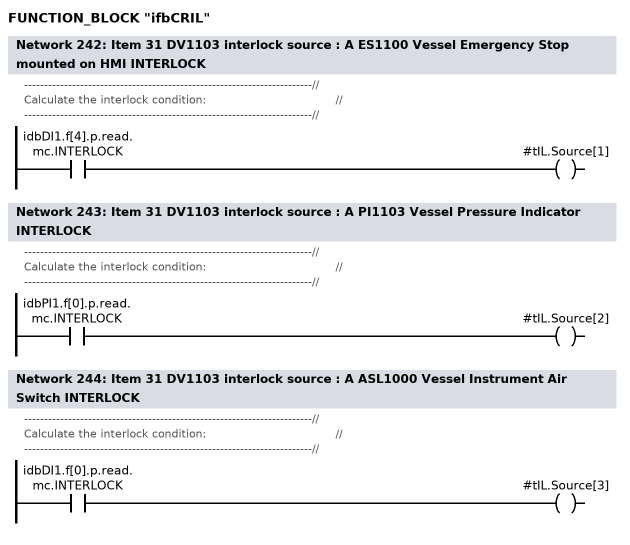
    A idbDI1.f[4].p.read.mc.INTERLOCK;
    = #tIL.Source[1];

NETWORK
TITLE = Item 31 DV1103 interlock source : A PI1103 Vessel Pressure Indicator INTERLOCK
    //------------------------------------------------------------------------//
    // Calculate the interlock condition:                                     //
    //------------------------------------------------------------------------//
    A idbPI1.f[0].p.read.mc.INTERLOCK;
    = #tIL.Source[2];

NETWORK
TITLE = Item 31 DV1103 interlock source : A ASL1000 Vessel Instrument Air Switch INTERLOCK
    //------------------------------------------------------------------------//
    // Calculate the interlock condition:                                     //
    //------------------------------------------------------------------------//
    A idbDI1.f[0].p.read.mc.INTERLOCK;
    = #tIL.Source[3];

NETWORK
TITLE = Item 31 DV1103 interlock source : AN ZSC1101 Vessel Manway Closed Indicator CLOSED
    //------------------------------------------------------------------------//
    // Calculate the interlock condition:                                     //
    //------------------------------------------------------------------------//
    AN(;
    L "idbZSC1".f[0].p.read.mc.STATE;
    L "dbCONST".BLK.ZSC1.STATE.CLOSED;
    ==I;
    );
    = #tIL.Source[4];

NETWORK
TITLE = Item 31 DV1103 interlock source : A ES1101 Mx Emergency Stop mounted on M1/M2 Shared HMI INTERLOCK
    //------------------------------------------------------------------------//
    // Calculate the interlock condition:                                     //
    //------------------------------------------------------------------------//
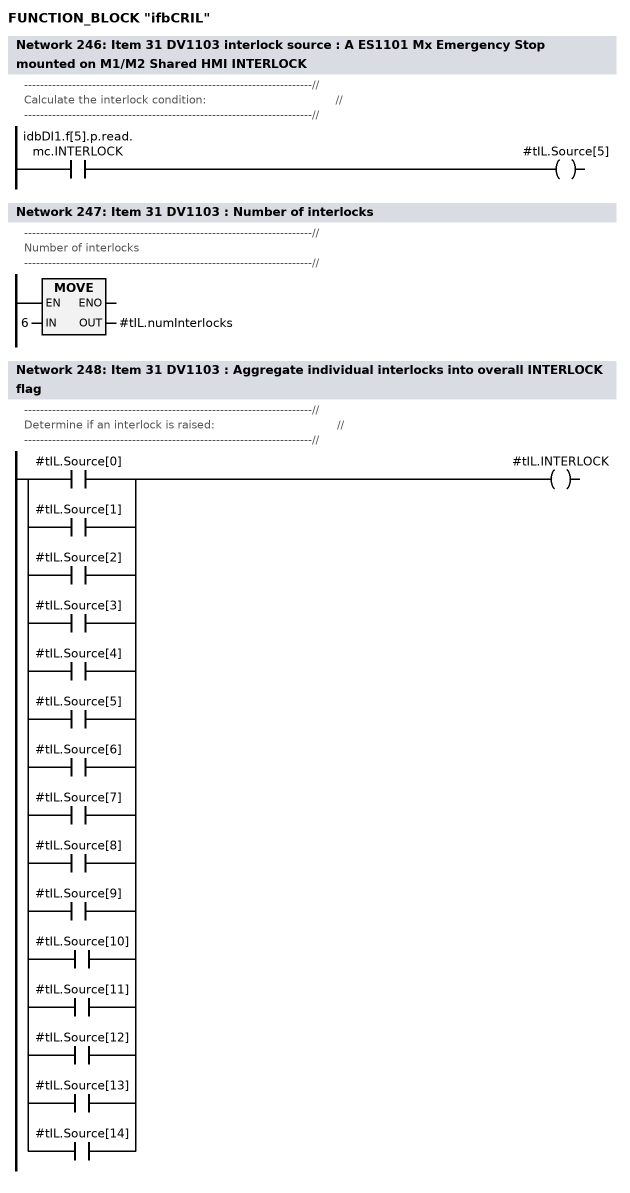
    A idbDI1.f[5].p.read.mc.INTERLOCK;
    = #tIL.Source[5];


NETWORK
TITLE = Item 31 DV1103 : Number of interlocks
    //------------------------------------------------------------------------//
    // Number of interlocks
    //------------------------------------------------------------------------//
    L 6;
    T #tIL.numInterlocks;

NETWORK
TITLE = Item 31 DV1103 : Aggregate individual interlocks into overall INTERLOCK flag
    //------------------------------------------------------------------------//
    // Determine if an interlock is raised:                                   //
    //------------------------------------------------------------------------//
    O #tIL.Source[0];
    O #tIL.Source[1];
    O #tIL.Source[2];
    O #tIL.Source[3];
    O #tIL.Source[4];
    O #tIL.Source[5];
    O #tIL.Source[6];
    O #tIL.Source[7];
    O #tIL.Source[8];
    O #tIL.Source[9];
    O #tIL.Source[10];
    O #tIL.Source[11];
    O #tIL.Source[12];
    O #tIL.Source[13];
    O #tIL.Source[14];
    = #tIL.INTERLOCK;

NETWORK
TITLE = Item 31 DV1103 : Update the instance data
    //------------------------------------------------------------------------//
    // Update the instance DB with the calculated interlock flags:            //
    //------------------------------------------------------------------------//
    CALL MOVE
    {value_type := 'Variant'}
    (   IN                   := #tIL ,
        OUT                  := #p[31]
    );

NETWORK
TITLE = Item 32 DV1105 : LP CA Supply Valve initialise variables
    //------------------------------------------------------------------------//
    // CRITICAL INTERLOCK   CRITICAL INTERLOCK   CRITICAL INTERLOCK   CRITICA //
    // CRITICAL INTERLOCK   CRITICAL INTERLOCK   CRITICAL INTERLOCK   CRITICA //
    //                                                                        //
    // Clear the interlock flag:                                              //
    //------------------------------------------------------------------------//
    A "alwaysLow";
    = #tIL.INTERLOCK;

    //------------------------------------------------------------------------//
    // Clear all interlock values to initialise them to off:                  //
    //------------------------------------------------------------------------//
    CALL FILL_BLK
    {value_type := 'Bool', count_type := 'UInt'}
    (   IN                   := 0 ,
        COUNT                := 15 ,
        OUT                  := #tIL.Source[0]
    );


NETWORK
TITLE = Item 32 DV1105 interlock source : A RD1101 Vessel Burst Disc ALARM
    //------------------------------------------------------------------------//
    // Calculate the interlock condition:                                     //
    //------------------------------------------------------------------------//
    A idbDI1.f[13].p.read.mc.INTERLOCK;
    = #tIL.Source[0];

NETWORK
TITLE = Item 32 DV1105 interlock source : A ES1100 Vessel Emergency Stop mounted on HMI INTERLOCK
    //------------------------------------------------------------------------//
    // Calculate the interlock condition:                                     //
    //------------------------------------------------------------------------//
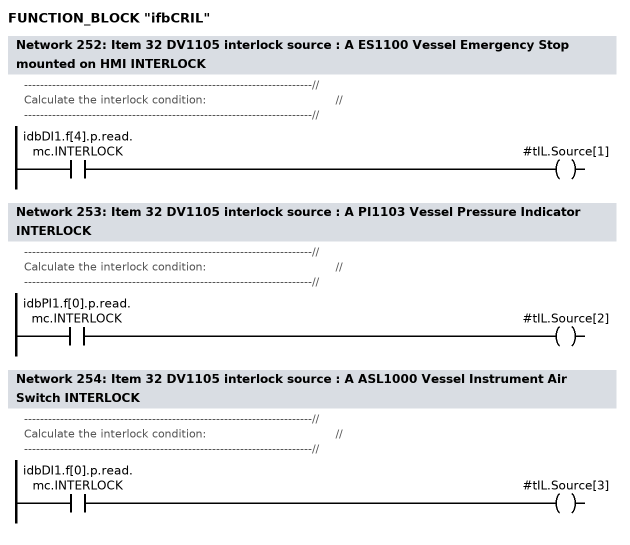
    A idbDI1.f[4].p.read.mc.INTERLOCK;
    = #tIL.Source[1];

NETWORK
TITLE = Item 32 DV1105 interlock source : A PI1103 Vessel Pressure Indicator INTERLOCK
    //------------------------------------------------------------------------//
    // Calculate the interlock condition:                                     //
    //------------------------------------------------------------------------//
    A idbPI1.f[0].p.read.mc.INTERLOCK;
    = #tIL.Source[2];

NETWORK
TITLE = Item 32 DV1105 interlock source : A ASL1000 Vessel Instrument Air Switch INTERLOCK
    //------------------------------------------------------------------------//
    // Calculate the interlock condition:                                     //
    //------------------------------------------------------------------------//
    A idbDI1.f[0].p.read.mc.INTERLOCK;
    = #tIL.Source[3];

NETWORK
TITLE = Item 32 DV1105 interlock source : AN ZSC1101 Vessel Manway Closed Indicator CLOSED
    //------------------------------------------------------------------------//
    // Calculate the interlock condition:                                     //
    //------------------------------------------------------------------------//
    AN(;
    L "idbZSC1".f[0].p.read.mc.STATE;
    L "dbCONST".BLK.ZSC1.STATE.CLOSED;
    ==I;
    );
    = #tIL.Source[4];

NETWORK
TITLE = Item 32 DV1105 interlock source : A ES1101 Mx Emergency Stop mounted on M1/M2 Shared HMI INTERLOCK
    //------------------------------------------------------------------------//
    // Calculate the interlock condition:                                     //
    //------------------------------------------------------------------------//
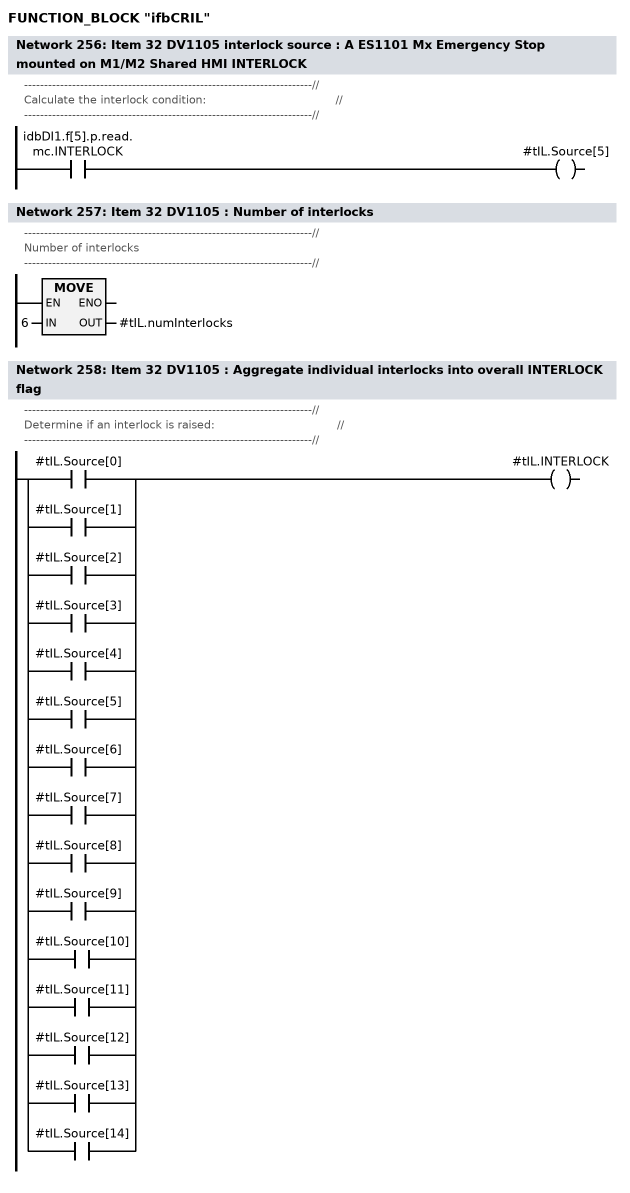
    A idbDI1.f[5].p.read.mc.INTERLOCK;
    = #tIL.Source[5];


NETWORK
TITLE = Item 32 DV1105 : Number of interlocks
    //------------------------------------------------------------------------//
    // Number of interlocks
    //------------------------------------------------------------------------//
    L 6;
    T #tIL.numInterlocks;

NETWORK
TITLE = Item 32 DV1105 : Aggregate individual interlocks into overall INTERLOCK flag
    //------------------------------------------------------------------------//
    // Determine if an interlock is raised:                                   //
    //------------------------------------------------------------------------//
    O #tIL.Source[0];
    O #tIL.Source[1];
    O #tIL.Source[2];
    O #tIL.Source[3];
    O #tIL.Source[4];
    O #tIL.Source[5];
    O #tIL.Source[6];
    O #tIL.Source[7];
    O #tIL.Source[8];
    O #tIL.Source[9];
    O #tIL.Source[10];
    O #tIL.Source[11];
    O #tIL.Source[12];
    O #tIL.Source[13];
    O #tIL.Source[14];
    = #tIL.INTERLOCK;

NETWORK
TITLE = Item 32 DV1105 : Update the instance data
    //------------------------------------------------------------------------//
    // Update the instance DB with the calculated interlock flags:            //
    //------------------------------------------------------------------------//
    CALL MOVE
    {value_type := 'Variant'}
    (   IN                   := #tIL ,
        OUT                  := #p[32]
    );

NETWORK
TITLE = Item 33 DV1107 : Vacuum valve initialise variables
    //------------------------------------------------------------------------//
    // CRITICAL INTERLOCK   CRITICAL INTERLOCK   CRITICAL INTERLOCK   CRITICA //
    // CRITICAL INTERLOCK   CRITICAL INTERLOCK   CRITICAL INTERLOCK   CRITICA //
    //                                                                        //
    // Clear the interlock flag:                                              //
    //------------------------------------------------------------------------//
    A "alwaysLow";
    = #tIL.INTERLOCK;

    //------------------------------------------------------------------------//
    // Clear all interlock values to initialise them to off:                  //
    //------------------------------------------------------------------------//
    CALL FILL_BLK
    {value_type := 'Bool', count_type := 'UInt'}
    (   IN                   := 0 ,
        COUNT                := 15 ,
        OUT                  := #tIL.Source[0]
    );


NETWORK
TITLE = Item 33 DV1107 interlock source : A RD1101 Vessel Burst Disc ALARM
    //------------------------------------------------------------------------//
    // Calculate the interlock condition:                                     //
    //------------------------------------------------------------------------//
    A idbDI1.f[13].p.read.mc.INTERLOCK;
    = #tIL.Source[0];

NETWORK
TITLE = Item 33 DV1107 interlock source : A ES1100 Vessel Emergency Stop mounted on HMI INTERLOCK
    //------------------------------------------------------------------------//
    // Calculate the interlock condition:                                     //
    //------------------------------------------------------------------------//
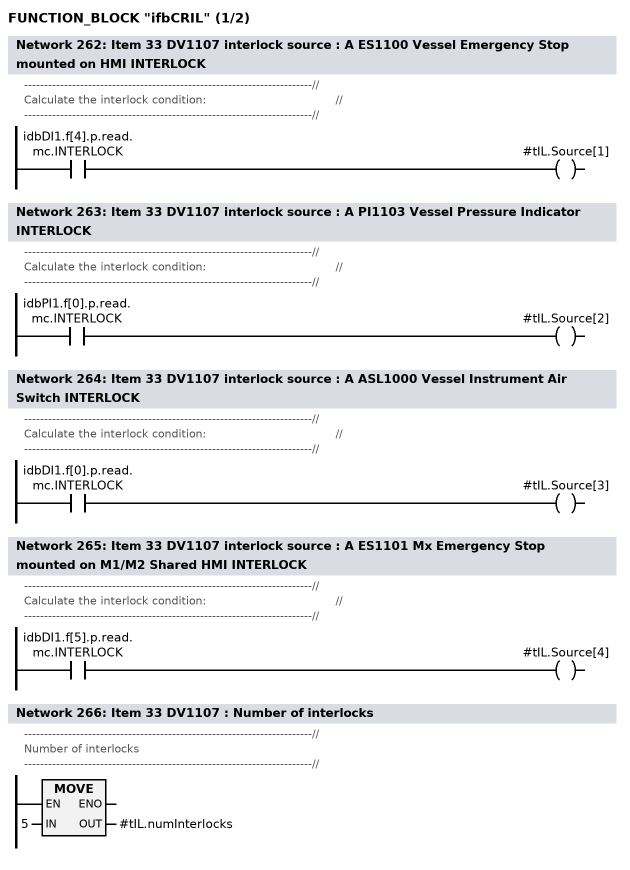
    A idbDI1.f[4].p.read.mc.INTERLOCK;
    = #tIL.Source[1];

NETWORK
TITLE = Item 33 DV1107 interlock source : A PI1103 Vessel Pressure Indicator INTERLOCK
    //------------------------------------------------------------------------//
    // Calculate the interlock condition:                                     //
    //------------------------------------------------------------------------//
    A idbPI1.f[0].p.read.mc.INTERLOCK;
    = #tIL.Source[2];

NETWORK
TITLE = Item 33 DV1107 interlock source : A ASL1000 Vessel Instrument Air Switch INTERLOCK
    //------------------------------------------------------------------------//
    // Calculate the interlock condition:                                     //
    //------------------------------------------------------------------------//
    A idbDI1.f[0].p.read.mc.INTERLOCK;
    = #tIL.Source[3];

NETWORK
TITLE = Item 33 DV1107 interlock source : A ES1101 Mx Emergency Stop mounted on M1/M2 Shared HMI INTERLOCK
    //------------------------------------------------------------------------//
    // Calculate the interlock condition:                                     //
    //------------------------------------------------------------------------//
    A idbDI1.f[5].p.read.mc.INTERLOCK;
    = #tIL.Source[4];


NETWORK
TITLE = Item 33 DV1107 : Number of interlocks
    //------------------------------------------------------------------------//
    // Number of interlocks
    //------------------------------------------------------------------------//
    L 5;
    T #tIL.numInterlocks;

NETWORK
TITLE = Item 33 DV1107 : Aggregate individual interlocks into overall INTERLOCK flag
    //------------------------------------------------------------------------//
    // Determine if an interlock is raised:                                   //
    //------------------------------------------------------------------------//
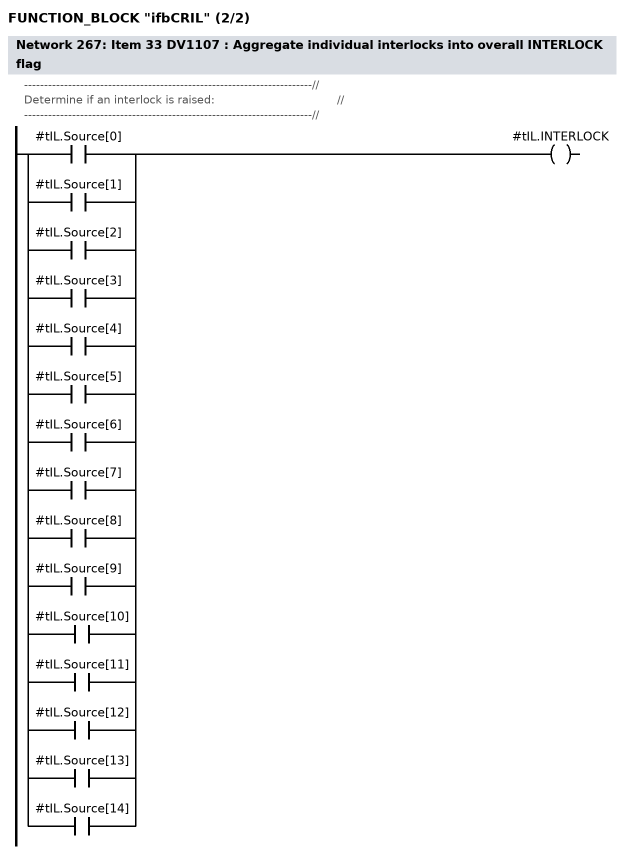
    O #tIL.Source[0];
    O #tIL.Source[1];
    O #tIL.Source[2];
    O #tIL.Source[3];
    O #tIL.Source[4];
    O #tIL.Source[5];
    O #tIL.Source[6];
    O #tIL.Source[7];
    O #tIL.Source[8];
    O #tIL.Source[9];
    O #tIL.Source[10];
    O #tIL.Source[11];
    O #tIL.Source[12];
    O #tIL.Source[13];
    O #tIL.Source[14];
    = #tIL.INTERLOCK;

NETWORK
TITLE = Item 33 DV1107 : Update the instance data
    //------------------------------------------------------------------------//
    // Update the instance DB with the calculated interlock flags:            //
    //------------------------------------------------------------------------//
    CALL MOVE
    {value_type := 'Variant'}
    (   IN                   := #tIL ,
        OUT                  := #p[33]
    );

NETWORK
TITLE = Item 34 DV1109 : PS Supply for WFI Loop initialise variables
    //------------------------------------------------------------------------//
    // CRITICAL INTERLOCK   CRITICAL INTERLOCK   CRITICAL INTERLOCK   CRITICA //
    // CRITICAL INTERLOCK   CRITICAL INTERLOCK   CRITICAL INTERLOCK   CRITICA //
    //                                                                        //
    // Clear the interlock flag:                                              //
    //------------------------------------------------------------------------//
    A "alwaysLow";
    = #tIL.INTERLOCK;

    //------------------------------------------------------------------------//
    // Clear all interlock values to initialise them to off:                  //
    //------------------------------------------------------------------------//
    CALL FILL_BLK
    {value_type := 'Bool', count_type := 'UInt'}
    (   IN                   := 0 ,
        COUNT                := 15 ,
        OUT                  := #tIL.Source[0]
    );


NETWORK
TITLE = Item 34 DV1109 interlock source : ON ZSC1107 Vessel inlet line Flowpath Indicator IN   ON ZSC1103 Vessel WFI Supply Flowpath Indicator IN
    //------------------------------------------------------------------------//
    // Calculate the interlock condition:                                     //
    //------------------------------------------------------------------------//
    ON(;
    L "idbZSC2".f[2].p.read.mc.STATE;
    L "dbCONST".BLK.ZSC2.STATE.IN;
    ==I;
    );
ON(;
    L "idbZSC2".f[0].p.read.mc.STATE;
    L "dbCONST".BLK.ZSC2.STATE.IN;
    ==I;
    );
    = #tIL.Source[0];

NETWORK
TITLE = Item 34 DV1109 interlock source : A DV1111 Vessel WFI Supply Valve OPENED
    //------------------------------------------------------------------------//
    // Calculate the interlock condition:                                     //
    //------------------------------------------------------------------------//
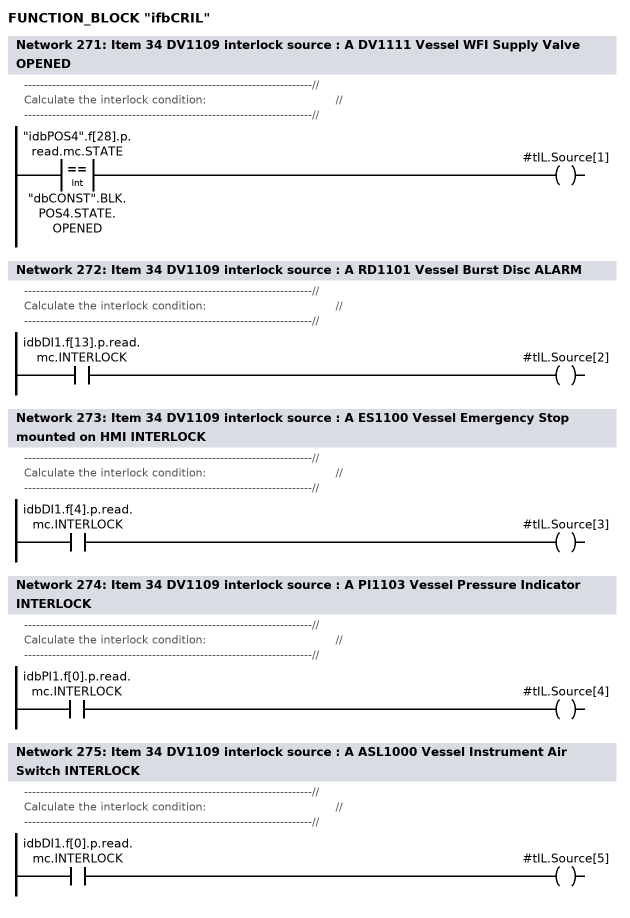
    A(;
    L "idbPOS4".f[28].p.read.mc.STATE;
    L "dbCONST".BLK.POS4.STATE.OPENED;
    ==I;
    );
    = #tIL.Source[1];

NETWORK
TITLE = Item 34 DV1109 interlock source : A RD1101 Vessel Burst Disc ALARM
    //------------------------------------------------------------------------//
    // Calculate the interlock condition:                                     //
    //------------------------------------------------------------------------//
    A idbDI1.f[13].p.read.mc.INTERLOCK;
    = #tIL.Source[2];

NETWORK
TITLE = Item 34 DV1109 interlock source : A ES1100 Vessel Emergency Stop mounted on HMI INTERLOCK
    //------------------------------------------------------------------------//
    // Calculate the interlock condition:                                     //
    //------------------------------------------------------------------------//
    A idbDI1.f[4].p.read.mc.INTERLOCK;
    = #tIL.Source[3];

NETWORK
TITLE = Item 34 DV1109 interlock source : A PI1103 Vessel Pressure Indicator INTERLOCK
    //------------------------------------------------------------------------//
    // Calculate the interlock condition:                                     //
    //------------------------------------------------------------------------//
    A idbPI1.f[0].p.read.mc.INTERLOCK;
    = #tIL.Source[4];

NETWORK
TITLE = Item 34 DV1109 interlock source : A ASL1000 Vessel Instrument Air Switch INTERLOCK
    //------------------------------------------------------------------------//
    // Calculate the interlock condition:                                     //
    //------------------------------------------------------------------------//
    A idbDI1.f[0].p.read.mc.INTERLOCK;
    = #tIL.Source[5];

NETWORK
TITLE = Item 34 DV1109 interlock source : AN ZSC1101 Vessel Manway Closed Indicator CLOSED
    //------------------------------------------------------------------------//
    // Calculate the interlock condition:                                     //
    //------------------------------------------------------------------------//
    AN(;
    L "idbZSC1".f[0].p.read.mc.STATE;
    L "dbCONST".BLK.ZSC1.STATE.CLOSED;
    ==I;
    );
    = #tIL.Source[6];

NETWORK
TITLE = Item 34 DV1109 interlock source : O MI1101 Mx Mass Indicator High High Alarm ALARM_HH   ON MI1101 Mx Mass Indicator Bad DQ DQ
    //------------------------------------------------------------------------//
    // Calculate the interlock condition:                                     //
    //------------------------------------------------------------------------//
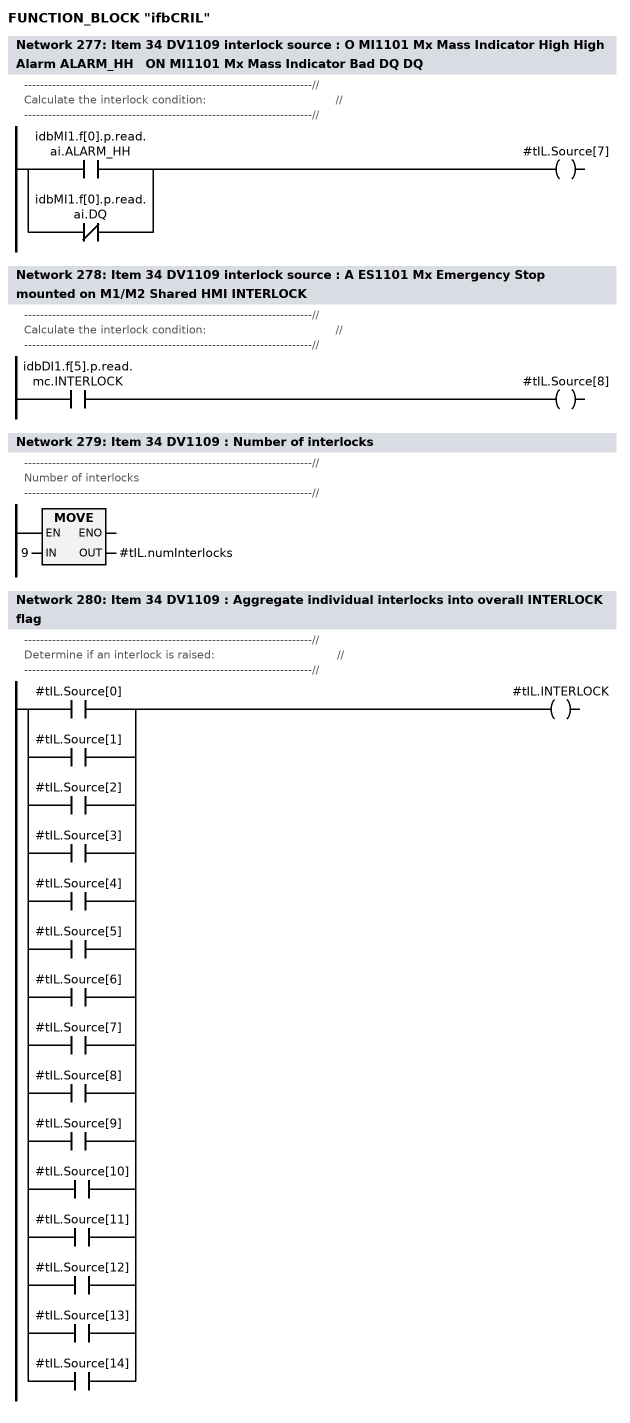
    O idbMI1.f[0].p.read.ai.ALARM_HH;
ON idbMI1.f[0].p.read.ai.DQ;
    = #tIL.Source[7];

NETWORK
TITLE = Item 34 DV1109 interlock source : A ES1101 Mx Emergency Stop mounted on M1/M2 Shared HMI INTERLOCK
    //------------------------------------------------------------------------//
    // Calculate the interlock condition:                                     //
    //------------------------------------------------------------------------//
    A idbDI1.f[5].p.read.mc.INTERLOCK;
    = #tIL.Source[8];


NETWORK
TITLE = Item 34 DV1109 : Number of interlocks
    //------------------------------------------------------------------------//
    // Number of interlocks
    //------------------------------------------------------------------------//
    L 9;
    T #tIL.numInterlocks;

NETWORK
TITLE = Item 34 DV1109 : Aggregate individual interlocks into overall INTERLOCK flag
    //------------------------------------------------------------------------//
    // Determine if an interlock is raised:                                   //
    //------------------------------------------------------------------------//
    O #tIL.Source[0];
    O #tIL.Source[1];
    O #tIL.Source[2];
    O #tIL.Source[3];
    O #tIL.Source[4];
    O #tIL.Source[5];
    O #tIL.Source[6];
    O #tIL.Source[7];
    O #tIL.Source[8];
    O #tIL.Source[9];
    O #tIL.Source[10];
    O #tIL.Source[11];
    O #tIL.Source[12];
    O #tIL.Source[13];
    O #tIL.Source[14];
    = #tIL.INTERLOCK;

NETWORK
TITLE = Item 34 DV1109 : Update the instance data
    //------------------------------------------------------------------------//
    // Update the instance DB with the calculated interlock flags:            //
    //------------------------------------------------------------------------//
    CALL MOVE
    {value_type := 'Variant'}
    (   IN                   := #tIL ,
        OUT                  := #p[34]
    );

NETWORK
TITLE = Item 35 DV1111 : WFI Supply Valve initialise variables
    //------------------------------------------------------------------------//
    // CRITICAL INTERLOCK   CRITICAL INTERLOCK   CRITICAL INTERLOCK   CRITICA //
    // CRITICAL INTERLOCK   CRITICAL INTERLOCK   CRITICAL INTERLOCK   CRITICA //
    //                                                                        //
    // Clear the interlock flag:                                              //
    //------------------------------------------------------------------------//
    A "alwaysLow";
    = #tIL.INTERLOCK;

    //------------------------------------------------------------------------//
    // Clear all interlock values to initialise them to off:                  //
    //------------------------------------------------------------------------//
    CALL FILL_BLK
    {value_type := 'Bool', count_type := 'UInt'}
    (   IN                   := 0 ,
        COUNT                := 15 ,
        OUT                  := #tIL.Source[0]
    );


NETWORK
TITLE = Item 35 DV1111 interlock source : ON ZSC1107 Vessel inlet line Flowpath Indicator IN   ON ZSC1103 Vessel WFI Supply Flowpath Indicator IN
    //------------------------------------------------------------------------//
    // Calculate the interlock condition:                                     //
    //------------------------------------------------------------------------//
    ON(;
    L "idbZSC2".f[2].p.read.mc.STATE;
    L "dbCONST".BLK.ZSC2.STATE.IN;
    ==I;
    );
ON(;
    L "idbZSC2".f[0].p.read.mc.STATE;
    L "dbCONST".BLK.ZSC2.STATE.IN;
    ==I;
    );
    = #tIL.Source[0];

NETWORK
TITLE = Item 35 DV1111 interlock source : A DV1109 Vessel PS Supply for WFI Loop OPENED
    //------------------------------------------------------------------------//
    // Calculate the interlock condition:                                     //
    //------------------------------------------------------------------------//
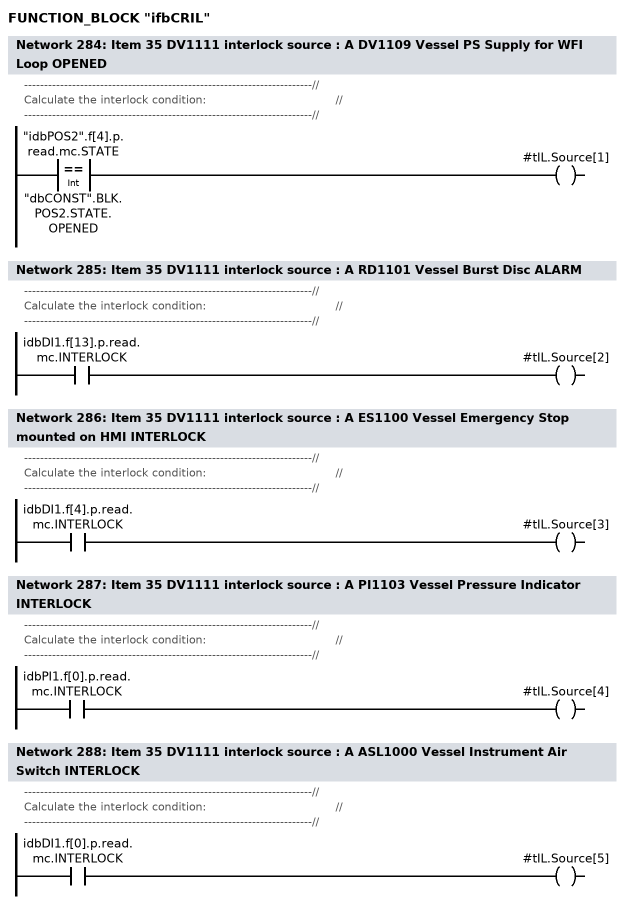
    A(;
    L "idbPOS2".f[4].p.read.mc.STATE;
    L "dbCONST".BLK.POS2.STATE.OPENED;
    ==I;
    );
    = #tIL.Source[1];

NETWORK
TITLE = Item 35 DV1111 interlock source : A RD1101 Vessel Burst Disc ALARM
    //------------------------------------------------------------------------//
    // Calculate the interlock condition:                                     //
    //------------------------------------------------------------------------//
    A idbDI1.f[13].p.read.mc.INTERLOCK;
    = #tIL.Source[2];

NETWORK
TITLE = Item 35 DV1111 interlock source : A ES1100 Vessel Emergency Stop mounted on HMI INTERLOCK
    //------------------------------------------------------------------------//
    // Calculate the interlock condition:                                     //
    //------------------------------------------------------------------------//
    A idbDI1.f[4].p.read.mc.INTERLOCK;
    = #tIL.Source[3];

NETWORK
TITLE = Item 35 DV1111 interlock source : A PI1103 Vessel Pressure Indicator INTERLOCK
    //------------------------------------------------------------------------//
    // Calculate the interlock condition:                                     //
    //------------------------------------------------------------------------//
    A idbPI1.f[0].p.read.mc.INTERLOCK;
    = #tIL.Source[4];

NETWORK
TITLE = Item 35 DV1111 interlock source : A ASL1000 Vessel Instrument Air Switch INTERLOCK
    //------------------------------------------------------------------------//
    // Calculate the interlock condition:                                     //
    //------------------------------------------------------------------------//
    A idbDI1.f[0].p.read.mc.INTERLOCK;
    = #tIL.Source[5];

NETWORK
TITLE = Item 35 DV1111 interlock source : AN ZSC1101 Vessel Manway Closed Indicator CLOSED
    //------------------------------------------------------------------------//
    // Calculate the interlock condition:                                     //
    //------------------------------------------------------------------------//
    AN(;
    L "idbZSC1".f[0].p.read.mc.STATE;
    L "dbCONST".BLK.ZSC1.STATE.CLOSED;
    ==I;
    );
    = #tIL.Source[6];

NETWORK
TITLE = Item 35 DV1111 interlock source : O MI1101 Mx Mass Indicator High High Alarm ALARM_HH   ON MI1101 Mx Mass Indicator Bad DQ DQ
    //------------------------------------------------------------------------//
    // Calculate the interlock condition:                                     //
    //------------------------------------------------------------------------//
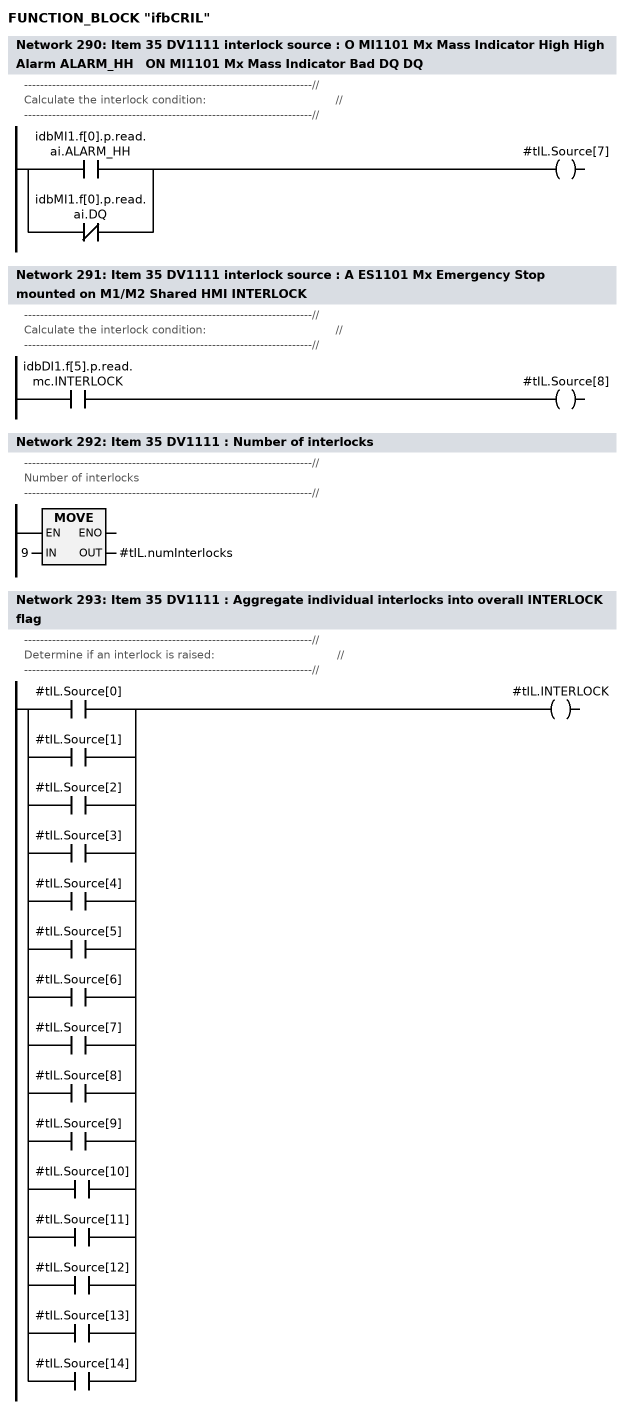
    O idbMI1.f[0].p.read.ai.ALARM_HH;
ON idbMI1.f[0].p.read.ai.DQ;
    = #tIL.Source[7];

NETWORK
TITLE = Item 35 DV1111 interlock source : A ES1101 Mx Emergency Stop mounted on M1/M2 Shared HMI INTERLOCK
    //------------------------------------------------------------------------//
    // Calculate the interlock condition:                                     //
    //------------------------------------------------------------------------//
    A idbDI1.f[5].p.read.mc.INTERLOCK;
    = #tIL.Source[8];


NETWORK
TITLE = Item 35 DV1111 : Number of interlocks
    //------------------------------------------------------------------------//
    // Number of interlocks
    //------------------------------------------------------------------------//
    L 9;
    T #tIL.numInterlocks;

NETWORK
TITLE = Item 35 DV1111 : Aggregate individual interlocks into overall INTERLOCK flag
    //------------------------------------------------------------------------//
    // Determine if an interlock is raised:                                   //
    //------------------------------------------------------------------------//
    O #tIL.Source[0];
    O #tIL.Source[1];
    O #tIL.Source[2];
    O #tIL.Source[3];
    O #tIL.Source[4];
    O #tIL.Source[5];
    O #tIL.Source[6];
    O #tIL.Source[7];
    O #tIL.Source[8];
    O #tIL.Source[9];
    O #tIL.Source[10];
    O #tIL.Source[11];
    O #tIL.Source[12];
    O #tIL.Source[13];
    O #tIL.Source[14];
    = #tIL.INTERLOCK;

NETWORK
TITLE = Item 35 DV1111 : Update the instance data
    //------------------------------------------------------------------------//
    // Update the instance DB with the calculated interlock flags:            //
    //------------------------------------------------------------------------//
    CALL MOVE
    {value_type := 'Variant'}
    (   IN                   := #tIL ,
        OUT                  := #p[35]
    );

NETWORK
TITLE = Item 36 DV1113 : PW Supply Valve initialise variables
    //------------------------------------------------------------------------//
    // CRITICAL INTERLOCK   CRITICAL INTERLOCK   CRITICAL INTERLOCK   CRITICA //
    // CRITICAL INTERLOCK   CRITICAL INTERLOCK   CRITICAL INTERLOCK   CRITICA //
    //                                                                        //
    // Clear the interlock flag:                                              //
    //------------------------------------------------------------------------//
    A "alwaysLow";
    = #tIL.INTERLOCK;

    //------------------------------------------------------------------------//
    // Clear all interlock values to initialise them to off:                  //
    //------------------------------------------------------------------------//
    CALL FILL_BLK
    {value_type := 'Bool', count_type := 'UInt'}
    (   IN                   := 0 ,
        COUNT                := 15 ,
        OUT                  := #tIL.Source[0]
    );


NETWORK
TITLE = Item 36 DV1113 interlock source : ON ZSC1107 Vessel inlet line Flowpath Indicator IN   ON ZSC1105 Vessel PW Supply Flowpath Indicator IN
    //------------------------------------------------------------------------//
    // Calculate the interlock condition:                                     //
    //------------------------------------------------------------------------//
    ON(;
    L "idbZSC2".f[2].p.read.mc.STATE;
    L "dbCONST".BLK.ZSC2.STATE.IN;
    ==I;
    );
ON(;
    L "idbZSC2".f[1].p.read.mc.STATE;
    L "dbCONST".BLK.ZSC2.STATE.IN;
    ==I;
    );
    = #tIL.Source[0];

NETWORK
TITLE = Item 36 DV1113 interlock source : A DV1115 Vessel PS Supply for PW Loop OPENED
    //------------------------------------------------------------------------//
    // Calculate the interlock condition:                                     //
    //------------------------------------------------------------------------//
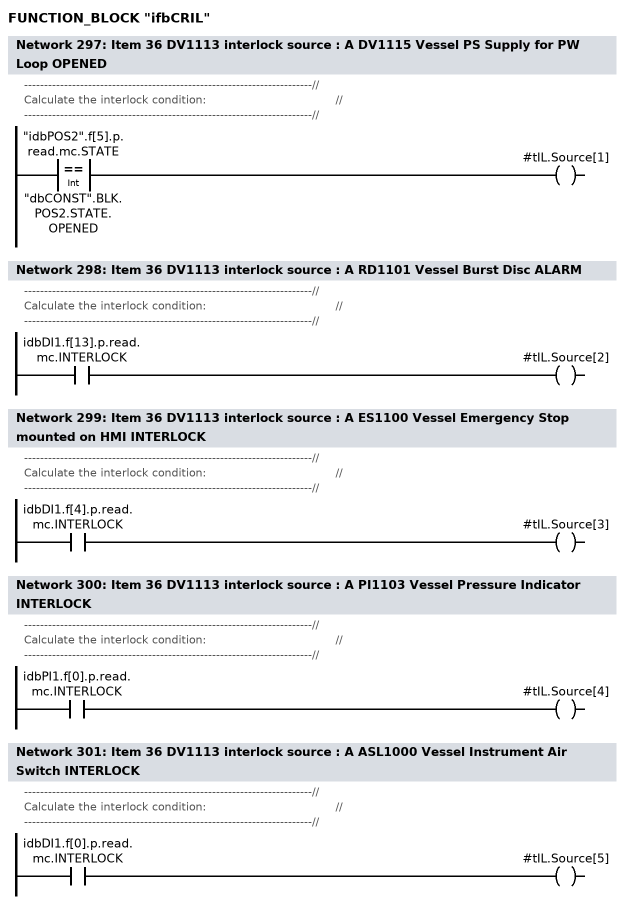
    A(;
    L "idbPOS2".f[5].p.read.mc.STATE;
    L "dbCONST".BLK.POS2.STATE.OPENED;
    ==I;
    );
    = #tIL.Source[1];

NETWORK
TITLE = Item 36 DV1113 interlock source : A RD1101 Vessel Burst Disc ALARM
    //------------------------------------------------------------------------//
    // Calculate the interlock condition:                                     //
    //------------------------------------------------------------------------//
    A idbDI1.f[13].p.read.mc.INTERLOCK;
    = #tIL.Source[2];

NETWORK
TITLE = Item 36 DV1113 interlock source : A ES1100 Vessel Emergency Stop mounted on HMI INTERLOCK
    //------------------------------------------------------------------------//
    // Calculate the interlock condition:                                     //
    //------------------------------------------------------------------------//
    A idbDI1.f[4].p.read.mc.INTERLOCK;
    = #tIL.Source[3];

NETWORK
TITLE = Item 36 DV1113 interlock source : A PI1103 Vessel Pressure Indicator INTERLOCK
    //------------------------------------------------------------------------//
    // Calculate the interlock condition:                                     //
    //------------------------------------------------------------------------//
    A idbPI1.f[0].p.read.mc.INTERLOCK;
    = #tIL.Source[4];

NETWORK
TITLE = Item 36 DV1113 interlock source : A ASL1000 Vessel Instrument Air Switch INTERLOCK
    //------------------------------------------------------------------------//
    // Calculate the interlock condition:                                     //
    //------------------------------------------------------------------------//
    A idbDI1.f[0].p.read.mc.INTERLOCK;
    = #tIL.Source[5];

NETWORK
TITLE = Item 36 DV1113 interlock source : AN ZSC1101 Vessel Manway Closed Indicator CLOSED
    //------------------------------------------------------------------------//
    // Calculate the interlock condition:                                     //
    //------------------------------------------------------------------------//
    AN(;
    L "idbZSC1".f[0].p.read.mc.STATE;
    L "dbCONST".BLK.ZSC1.STATE.CLOSED;
    ==I;
    );
    = #tIL.Source[6];

NETWORK
TITLE = Item 36 DV1113 interlock source : O MI1101 Mx Mass Indicator High High Alarm ALARM_HH   ON MI1101 Mx Mass Indicator Bad DQ DQ
    //------------------------------------------------------------------------//
    // Calculate the interlock condition:                                     //
    //------------------------------------------------------------------------//
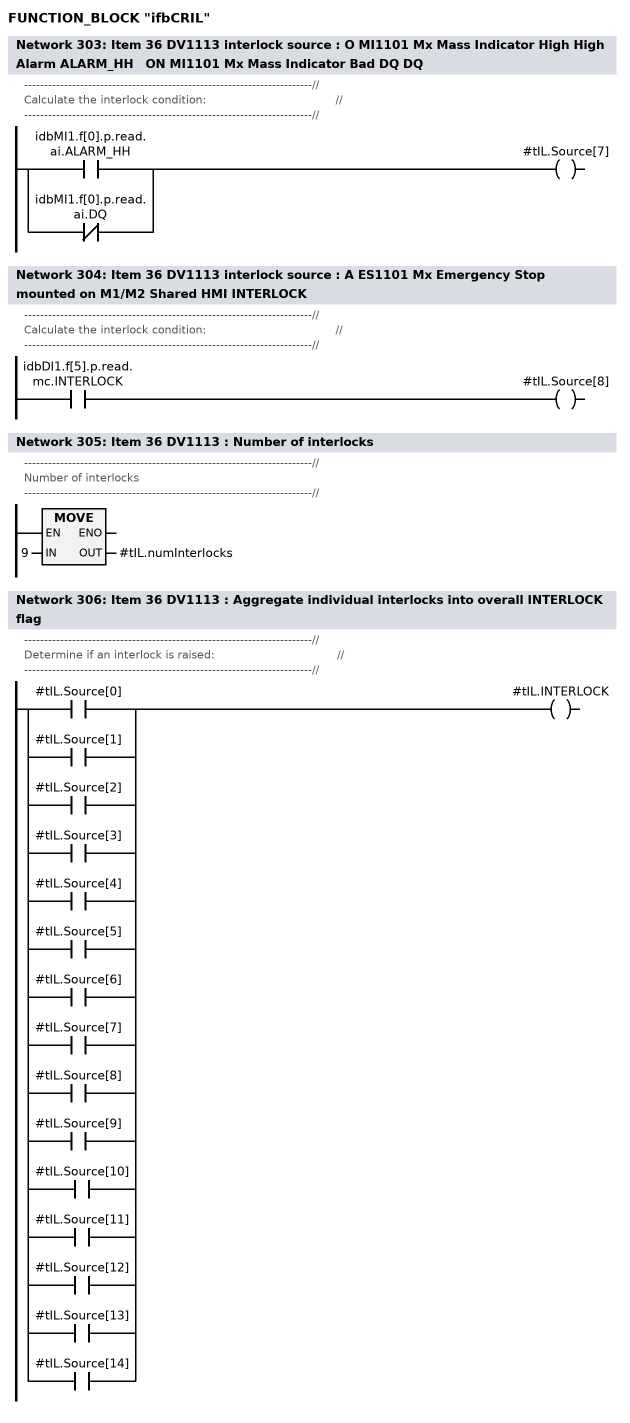
    O idbMI1.f[0].p.read.ai.ALARM_HH;
ON idbMI1.f[0].p.read.ai.DQ;
    = #tIL.Source[7];

NETWORK
TITLE = Item 36 DV1113 interlock source : A ES1101 Mx Emergency Stop mounted on M1/M2 Shared HMI INTERLOCK
    //------------------------------------------------------------------------//
    // Calculate the interlock condition:                                     //
    //------------------------------------------------------------------------//
    A idbDI1.f[5].p.read.mc.INTERLOCK;
    = #tIL.Source[8];


NETWORK
TITLE = Item 36 DV1113 : Number of interlocks
    //------------------------------------------------------------------------//
    // Number of interlocks
    //------------------------------------------------------------------------//
    L 9;
    T #tIL.numInterlocks;

NETWORK
TITLE = Item 36 DV1113 : Aggregate individual interlocks into overall INTERLOCK flag
    //------------------------------------------------------------------------//
    // Determine if an interlock is raised:                                   //
    //------------------------------------------------------------------------//
    O #tIL.Source[0];
    O #tIL.Source[1];
    O #tIL.Source[2];
    O #tIL.Source[3];
    O #tIL.Source[4];
    O #tIL.Source[5];
    O #tIL.Source[6];
    O #tIL.Source[7];
    O #tIL.Source[8];
    O #tIL.Source[9];
    O #tIL.Source[10];
    O #tIL.Source[11];
    O #tIL.Source[12];
    O #tIL.Source[13];
    O #tIL.Source[14];
    = #tIL.INTERLOCK;

NETWORK
TITLE = Item 36 DV1113 : Update the instance data
    //------------------------------------------------------------------------//
    // Update the instance DB with the calculated interlock flags:            //
    //------------------------------------------------------------------------//
    CALL MOVE
    {value_type := 'Variant'}
    (   IN                   := #tIL ,
        OUT                  := #p[36]
    );

NETWORK
TITLE = Item 37 DV1115 : PS Supply for PW Loop initialise variables
    //------------------------------------------------------------------------//
    // CRITICAL INTERLOCK   CRITICAL INTERLOCK   CRITICAL INTERLOCK   CRITICA //
    // CRITICAL INTERLOCK   CRITICAL INTERLOCK   CRITICAL INTERLOCK   CRITICA //
    //                                                                        //
    // Clear the interlock flag:                                              //
    //------------------------------------------------------------------------//
    A "alwaysLow";
    = #tIL.INTERLOCK;

    //------------------------------------------------------------------------//
    // Clear all interlock values to initialise them to off:                  //
    //------------------------------------------------------------------------//
    CALL FILL_BLK
    {value_type := 'Bool', count_type := 'UInt'}
    (   IN                   := 0 ,
        COUNT                := 15 ,
        OUT                  := #tIL.Source[0]
    );


NETWORK
TITLE = Item 37 DV1115 interlock source : ON ZSC1107 Vessel inlet line Flowpath Indicator IN   ON ZSC1105 Vessel PW Supply Flowpath Indicator IN
    //------------------------------------------------------------------------//
    // Calculate the interlock condition:                                     //
    //------------------------------------------------------------------------//
    ON(;
    L "idbZSC2".f[2].p.read.mc.STATE;
    L "dbCONST".BLK.ZSC2.STATE.IN;
    ==I;
    );
ON(;
    L "idbZSC2".f[1].p.read.mc.STATE;
    L "dbCONST".BLK.ZSC2.STATE.IN;
    ==I;
    );
    = #tIL.Source[0];

NETWORK
TITLE = Item 37 DV1115 interlock source : A DV1113 Vessel PW Supply Valve OPENED
    //------------------------------------------------------------------------//
    // Calculate the interlock condition:                                     //
    //------------------------------------------------------------------------//
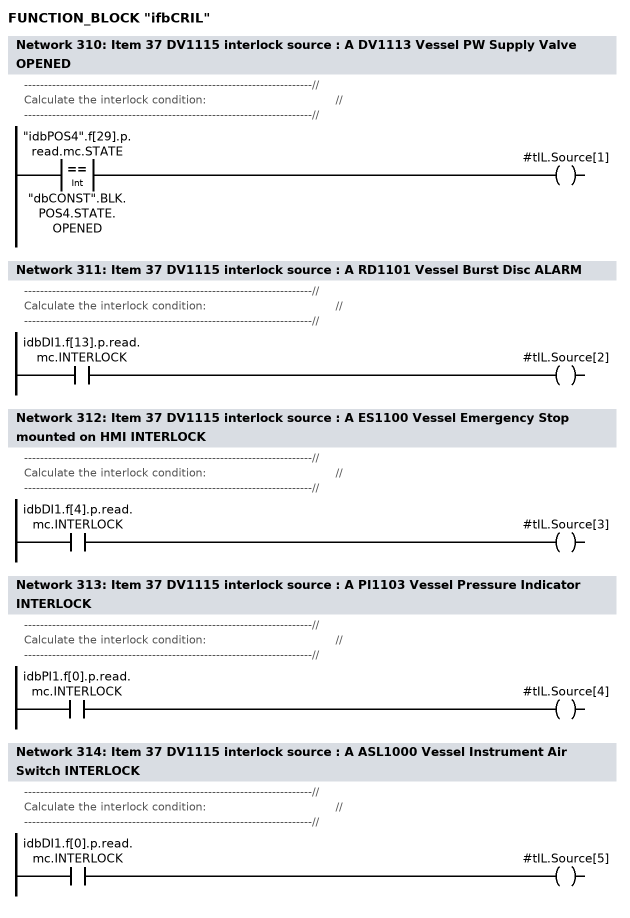
    A(;
    L "idbPOS4".f[29].p.read.mc.STATE;
    L "dbCONST".BLK.POS4.STATE.OPENED;
    ==I;
    );
    = #tIL.Source[1];

NETWORK
TITLE = Item 37 DV1115 interlock source : A RD1101 Vessel Burst Disc ALARM
    //------------------------------------------------------------------------//
    // Calculate the interlock condition:                                     //
    //------------------------------------------------------------------------//
    A idbDI1.f[13].p.read.mc.INTERLOCK;
    = #tIL.Source[2];

NETWORK
TITLE = Item 37 DV1115 interlock source : A ES1100 Vessel Emergency Stop mounted on HMI INTERLOCK
    //------------------------------------------------------------------------//
    // Calculate the interlock condition:                                     //
    //------------------------------------------------------------------------//
    A idbDI1.f[4].p.read.mc.INTERLOCK;
    = #tIL.Source[3];

NETWORK
TITLE = Item 37 DV1115 interlock source : A PI1103 Vessel Pressure Indicator INTERLOCK
    //------------------------------------------------------------------------//
    // Calculate the interlock condition:                                     //
    //------------------------------------------------------------------------//
    A idbPI1.f[0].p.read.mc.INTERLOCK;
    = #tIL.Source[4];

NETWORK
TITLE = Item 37 DV1115 interlock source : A ASL1000 Vessel Instrument Air Switch INTERLOCK
    //------------------------------------------------------------------------//
    // Calculate the interlock condition:                                     //
    //------------------------------------------------------------------------//
    A idbDI1.f[0].p.read.mc.INTERLOCK;
    = #tIL.Source[5];

NETWORK
TITLE = Item 37 DV1115 interlock source : AN ZSC1101 Vessel Manway Closed Indicator CLOSED
    //------------------------------------------------------------------------//
    // Calculate the interlock condition:                                     //
    //------------------------------------------------------------------------//
    AN(;
    L "idbZSC1".f[0].p.read.mc.STATE;
    L "dbCONST".BLK.ZSC1.STATE.CLOSED;
    ==I;
    );
    = #tIL.Source[6];

NETWORK
TITLE = Item 37 DV1115 interlock source : O MI1101 Mx Mass Indicator High High Alarm ALARM_HH   ON MI1101 Mx Mass Indicator Bad DQ DQ
    //------------------------------------------------------------------------//
    // Calculate the interlock condition:                                     //
    //------------------------------------------------------------------------//
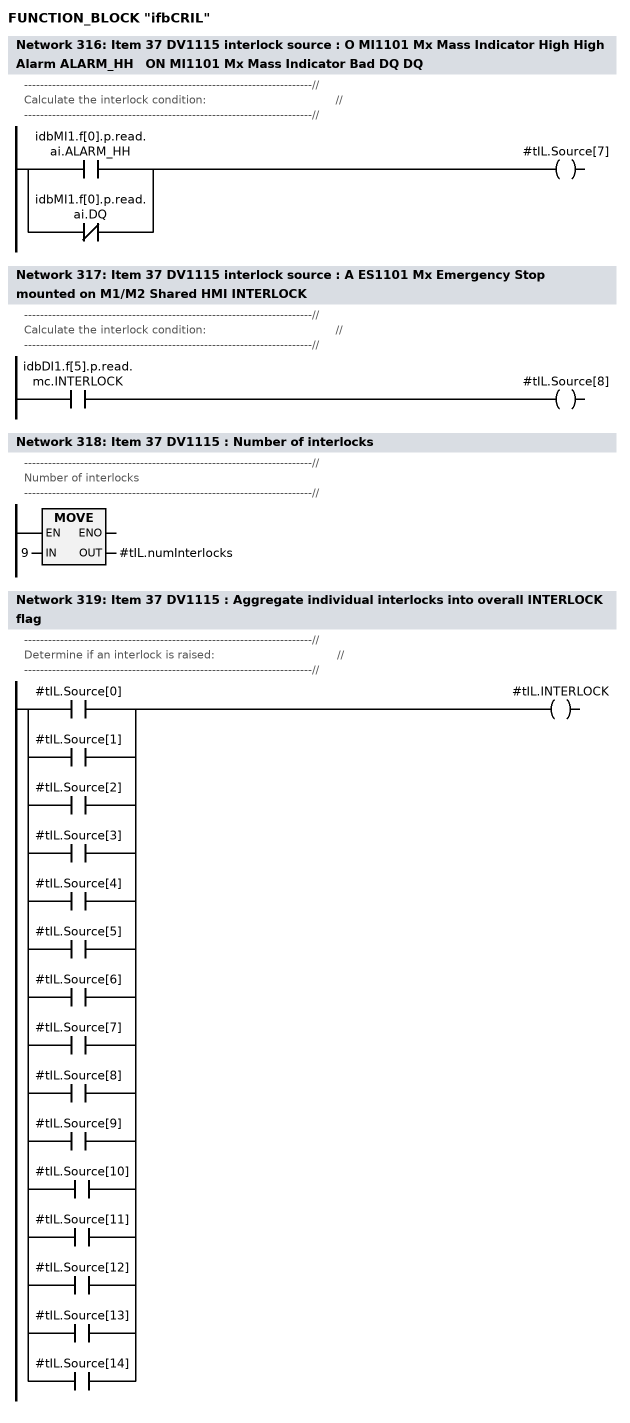
    O idbMI1.f[0].p.read.ai.ALARM_HH;
ON idbMI1.f[0].p.read.ai.DQ;
    = #tIL.Source[7];

NETWORK
TITLE = Item 37 DV1115 interlock source : A ES1101 Mx Emergency Stop mounted on M1/M2 Shared HMI INTERLOCK
    //------------------------------------------------------------------------//
    // Calculate the interlock condition:                                     //
    //------------------------------------------------------------------------//
    A idbDI1.f[5].p.read.mc.INTERLOCK;
    = #tIL.Source[8];


NETWORK
TITLE = Item 37 DV1115 : Number of interlocks
    //------------------------------------------------------------------------//
    // Number of interlocks
    //------------------------------------------------------------------------//
    L 9;
    T #tIL.numInterlocks;

NETWORK
TITLE = Item 37 DV1115 : Aggregate individual interlocks into overall INTERLOCK flag
    //------------------------------------------------------------------------//
    // Determine if an interlock is raised:                                   //
    //------------------------------------------------------------------------//
    O #tIL.Source[0];
    O #tIL.Source[1];
    O #tIL.Source[2];
    O #tIL.Source[3];
    O #tIL.Source[4];
    O #tIL.Source[5];
    O #tIL.Source[6];
    O #tIL.Source[7];
    O #tIL.Source[8];
    O #tIL.Source[9];
    O #tIL.Source[10];
    O #tIL.Source[11];
    O #tIL.Source[12];
    O #tIL.Source[13];
    O #tIL.Source[14];
    = #tIL.INTERLOCK;

NETWORK
TITLE = Item 37 DV1115 : Update the instance data
    //------------------------------------------------------------------------//
    // Update the instance DB with the calculated interlock flags:            //
    //------------------------------------------------------------------------//
    CALL MOVE
    {value_type := 'Variant'}
    (   IN                   := #tIL ,
        OUT                  := #p[37]
    );

NETWORK
TITLE = Item 38 DV1117 : Spray Ball 1 Valve initialise variables
    //------------------------------------------------------------------------//
    // CRITICAL INTERLOCK   CRITICAL INTERLOCK   CRITICAL INTERLOCK   CRITICA //
    // CRITICAL INTERLOCK   CRITICAL INTERLOCK   CRITICAL INTERLOCK   CRITICA //
    //                                                                        //
    // Clear the interlock flag:                                              //
    //------------------------------------------------------------------------//
    A "alwaysLow";
    = #tIL.INTERLOCK;

    //------------------------------------------------------------------------//
    // Clear all interlock values to initialise them to off:                  //
    //------------------------------------------------------------------------//
    CALL FILL_BLK
    {value_type := 'Bool', count_type := 'UInt'}
    (   IN                   := 0 ,
        COUNT                := 15 ,
        OUT                  := #tIL.Source[0]
    );


NETWORK
TITLE = Item 38 DV1117 interlock source : A RD1101 Vessel Burst Disc ALARM
    //------------------------------------------------------------------------//
    // Calculate the interlock condition:                                     //
    //------------------------------------------------------------------------//
    A idbDI1.f[13].p.read.mc.INTERLOCK;
    = #tIL.Source[0];

NETWORK
TITLE = Item 38 DV1117 interlock source : A ES1100 Vessel Emergency Stop mounted on HMI INTERLOCK
    //------------------------------------------------------------------------//
    // Calculate the interlock condition:                                     //
    //------------------------------------------------------------------------//
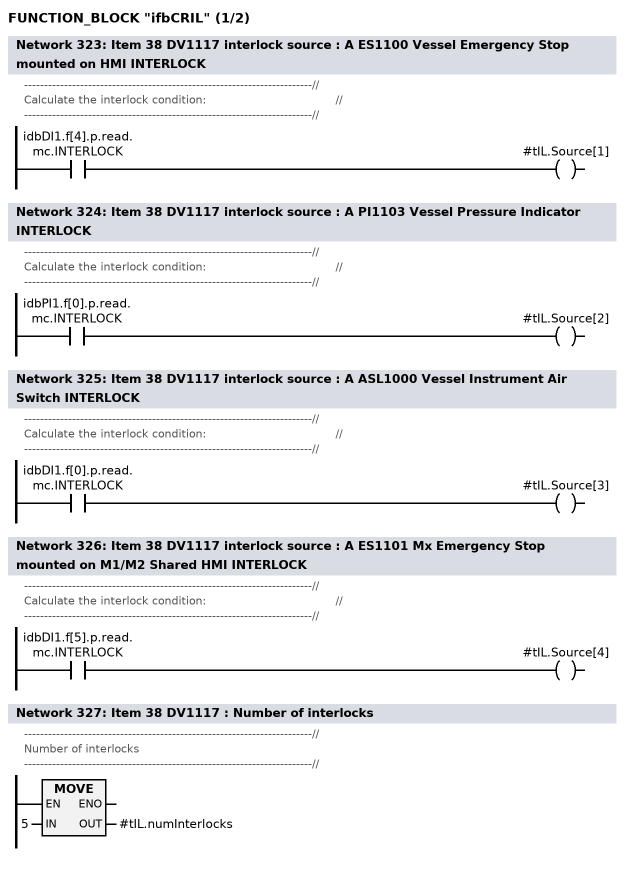
    A idbDI1.f[4].p.read.mc.INTERLOCK;
    = #tIL.Source[1];

NETWORK
TITLE = Item 38 DV1117 interlock source : A PI1103 Vessel Pressure Indicator INTERLOCK
    //------------------------------------------------------------------------//
    // Calculate the interlock condition:                                     //
    //------------------------------------------------------------------------//
    A idbPI1.f[0].p.read.mc.INTERLOCK;
    = #tIL.Source[2];

NETWORK
TITLE = Item 38 DV1117 interlock source : A ASL1000 Vessel Instrument Air Switch INTERLOCK
    //------------------------------------------------------------------------//
    // Calculate the interlock condition:                                     //
    //------------------------------------------------------------------------//
    A idbDI1.f[0].p.read.mc.INTERLOCK;
    = #tIL.Source[3];

NETWORK
TITLE = Item 38 DV1117 interlock source : A ES1101 Mx Emergency Stop mounted on M1/M2 Shared HMI INTERLOCK
    //------------------------------------------------------------------------//
    // Calculate the interlock condition:                                     //
    //------------------------------------------------------------------------//
    A idbDI1.f[5].p.read.mc.INTERLOCK;
    = #tIL.Source[4];


NETWORK
TITLE = Item 38 DV1117 : Number of interlocks
    //------------------------------------------------------------------------//
    // Number of interlocks
    //------------------------------------------------------------------------//
    L 5;
    T #tIL.numInterlocks;

NETWORK
TITLE = Item 38 DV1117 : Aggregate individual interlocks into overall INTERLOCK flag
    //------------------------------------------------------------------------//
    // Determine if an interlock is raised:                                   //
    //------------------------------------------------------------------------//
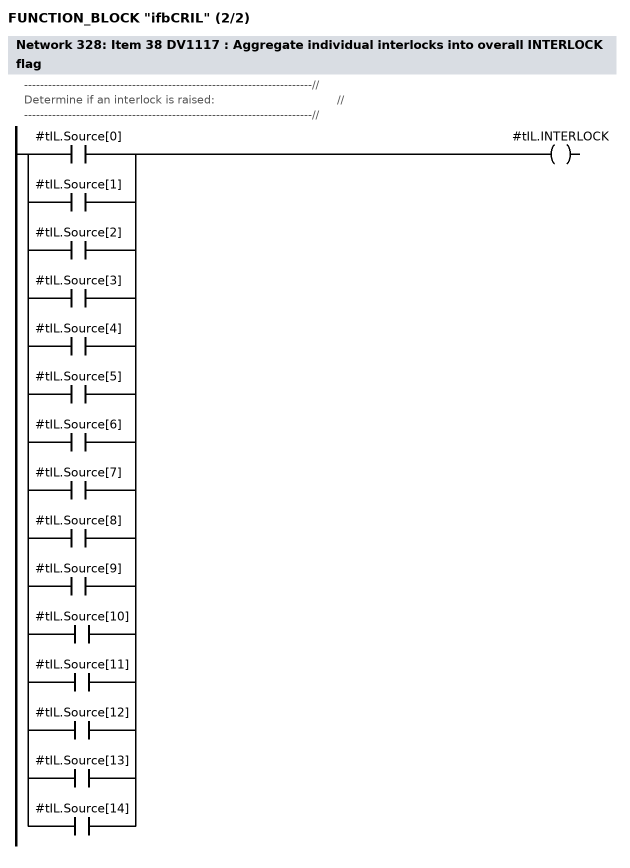
    O #tIL.Source[0];
    O #tIL.Source[1];
    O #tIL.Source[2];
    O #tIL.Source[3];
    O #tIL.Source[4];
    O #tIL.Source[5];
    O #tIL.Source[6];
    O #tIL.Source[7];
    O #tIL.Source[8];
    O #tIL.Source[9];
    O #tIL.Source[10];
    O #tIL.Source[11];
    O #tIL.Source[12];
    O #tIL.Source[13];
    O #tIL.Source[14];
    = #tIL.INTERLOCK;

NETWORK
TITLE = Item 38 DV1117 : Update the instance data
    //------------------------------------------------------------------------//
    // Update the instance DB with the calculated interlock flags:            //
    //------------------------------------------------------------------------//
    CALL MOVE
    {value_type := 'Variant'}
    (   IN                   := #tIL ,
        OUT                  := #p[38]
    );

NETWORK
TITLE = Item 39 DV1119 : Spray Ball 2 Valve initialise variables
    //------------------------------------------------------------------------//
    // CRITICAL INTERLOCK   CRITICAL INTERLOCK   CRITICAL INTERLOCK   CRITICA //
    // CRITICAL INTERLOCK   CRITICAL INTERLOCK   CRITICAL INTERLOCK   CRITICA //
    //                                                                        //
    // Clear the interlock flag:                                              //
    //------------------------------------------------------------------------//
    A "alwaysLow";
    = #tIL.INTERLOCK;

    //------------------------------------------------------------------------//
    // Clear all interlock values to initialise them to off:                  //
    //------------------------------------------------------------------------//
    CALL FILL_BLK
    {value_type := 'Bool', count_type := 'UInt'}
    (   IN                   := 0 ,
        COUNT                := 15 ,
        OUT                  := #tIL.Source[0]
    );


NETWORK
TITLE = Item 39 DV1119 interlock source : A RD1101 Vessel Burst Disc ALARM
    //------------------------------------------------------------------------//
    // Calculate the interlock condition:                                     //
    //------------------------------------------------------------------------//
    A idbDI1.f[13].p.read.mc.INTERLOCK;
    = #tIL.Source[0];

NETWORK
TITLE = Item 39 DV1119 interlock source : A ES1100 Vessel Emergency Stop mounted on HMI INTERLOCK
    //------------------------------------------------------------------------//
    // Calculate the interlock condition:                                     //
    //------------------------------------------------------------------------//
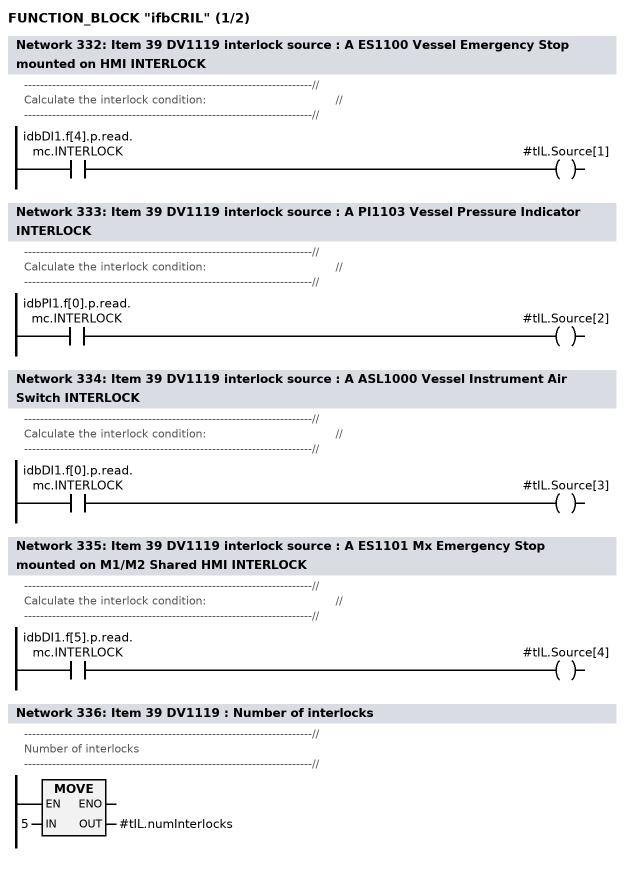
    A idbDI1.f[4].p.read.mc.INTERLOCK;
    = #tIL.Source[1];

NETWORK
TITLE = Item 39 DV1119 interlock source : A PI1103 Vessel Pressure Indicator INTERLOCK
    //------------------------------------------------------------------------//
    // Calculate the interlock condition:                                     //
    //------------------------------------------------------------------------//
    A idbPI1.f[0].p.read.mc.INTERLOCK;
    = #tIL.Source[2];

NETWORK
TITLE = Item 39 DV1119 interlock source : A ASL1000 Vessel Instrument Air Switch INTERLOCK
    //------------------------------------------------------------------------//
    // Calculate the interlock condition:                                     //
    //------------------------------------------------------------------------//
    A idbDI1.f[0].p.read.mc.INTERLOCK;
    = #tIL.Source[3];

NETWORK
TITLE = Item 39 DV1119 interlock source : A ES1101 Mx Emergency Stop mounted on M1/M2 Shared HMI INTERLOCK
    //------------------------------------------------------------------------//
    // Calculate the interlock condition:                                     //
    //------------------------------------------------------------------------//
    A idbDI1.f[5].p.read.mc.INTERLOCK;
    = #tIL.Source[4];


NETWORK
TITLE = Item 39 DV1119 : Number of interlocks
    //------------------------------------------------------------------------//
    // Number of interlocks
    //------------------------------------------------------------------------//
    L 5;
    T #tIL.numInterlocks;

NETWORK
TITLE = Item 39 DV1119 : Aggregate individual interlocks into overall INTERLOCK flag
    //------------------------------------------------------------------------//
    // Determine if an interlock is raised:                                   //
    //------------------------------------------------------------------------//
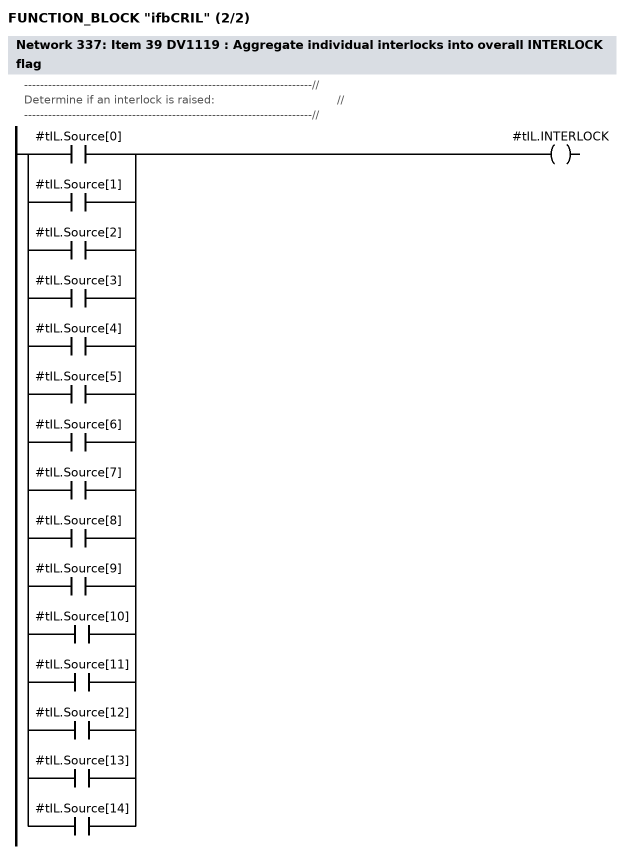
    O #tIL.Source[0];
    O #tIL.Source[1];
    O #tIL.Source[2];
    O #tIL.Source[3];
    O #tIL.Source[4];
    O #tIL.Source[5];
    O #tIL.Source[6];
    O #tIL.Source[7];
    O #tIL.Source[8];
    O #tIL.Source[9];
    O #tIL.Source[10];
    O #tIL.Source[11];
    O #tIL.Source[12];
    O #tIL.Source[13];
    O #tIL.Source[14];
    = #tIL.INTERLOCK;

NETWORK
TITLE = Item 39 DV1119 : Update the instance data
    //------------------------------------------------------------------------//
    // Update the instance DB with the calculated interlock flags:            //
    //------------------------------------------------------------------------//
    CALL MOVE
    {value_type := 'Variant'}
    (   IN                   := #tIL ,
        OUT                  := #p[39]
    );

NETWORK
TITLE = Item 40 DV1121 : Outlet Valve initialise variables
    //------------------------------------------------------------------------//
    // CRITICAL INTERLOCK   CRITICAL INTERLOCK   CRITICAL INTERLOCK   CRITICA //
    // CRITICAL INTERLOCK   CRITICAL INTERLOCK   CRITICAL INTERLOCK   CRITICA //
    //                                                                        //
    // Clear the interlock flag:                                              //
    //------------------------------------------------------------------------//
    A "alwaysLow";
    = #tIL.INTERLOCK;

    //------------------------------------------------------------------------//
    // Clear all interlock values to initialise them to off:                  //
    //------------------------------------------------------------------------//
    CALL FILL_BLK
    {value_type := 'Bool', count_type := 'UInt'}
    (   IN                   := 0 ,
        COUNT                := 15 ,
        OUT                  := #tIL.Source[0]
    );


NETWORK
TITLE = Item 40 DV1121 interlock source : A RD1101 Vessel Burst Disc ALARM
    //------------------------------------------------------------------------//
    // Calculate the interlock condition:                                     //
    //------------------------------------------------------------------------//
    A idbDI1.f[13].p.read.mc.INTERLOCK;
    = #tIL.Source[0];

NETWORK
TITLE = Item 40 DV1121 interlock source : A ES1100 Vessel Emergency Stop mounted on HMI INTERLOCK
    //------------------------------------------------------------------------//
    // Calculate the interlock condition:                                     //
    //------------------------------------------------------------------------//
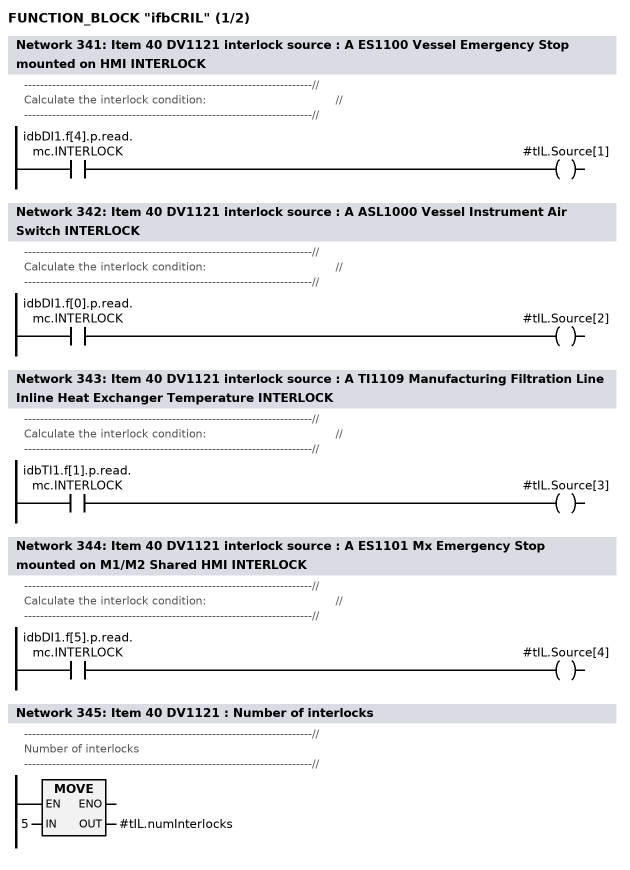
    A idbDI1.f[4].p.read.mc.INTERLOCK;
    = #tIL.Source[1];

NETWORK
TITLE = Item 40 DV1121 interlock source : A ASL1000 Vessel Instrument Air Switch INTERLOCK
    //------------------------------------------------------------------------//
    // Calculate the interlock condition:                                     //
    //------------------------------------------------------------------------//
    A idbDI1.f[0].p.read.mc.INTERLOCK;
    = #tIL.Source[2];

NETWORK
TITLE = Item 40 DV1121 interlock source : A TI1109 Manufacturing Filtration Line Inline Heat Exchanger Temperature INTERLOCK
    //------------------------------------------------------------------------//
    // Calculate the interlock condition:                                     //
    //------------------------------------------------------------------------//
    A idbTI1.f[1].p.read.mc.INTERLOCK;
    = #tIL.Source[3];

NETWORK
TITLE = Item 40 DV1121 interlock source : A ES1101 Mx Emergency Stop mounted on M1/M2 Shared HMI INTERLOCK
    //------------------------------------------------------------------------//
    // Calculate the interlock condition:                                     //
    //------------------------------------------------------------------------//
    A idbDI1.f[5].p.read.mc.INTERLOCK;
    = #tIL.Source[4];


NETWORK
TITLE = Item 40 DV1121 : Number of interlocks
    //------------------------------------------------------------------------//
    // Number of interlocks
    //------------------------------------------------------------------------//
    L 5;
    T #tIL.numInterlocks;

NETWORK
TITLE = Item 40 DV1121 : Aggregate individual interlocks into overall INTERLOCK flag
    //------------------------------------------------------------------------//
    // Determine if an interlock is raised:                                   //
    //------------------------------------------------------------------------//
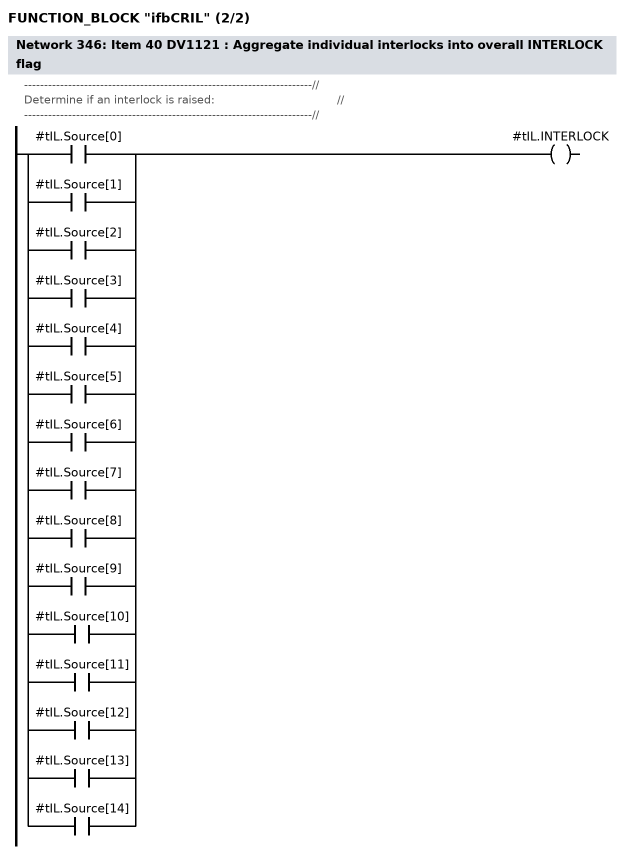
    O #tIL.Source[0];
    O #tIL.Source[1];
    O #tIL.Source[2];
    O #tIL.Source[3];
    O #tIL.Source[4];
    O #tIL.Source[5];
    O #tIL.Source[6];
    O #tIL.Source[7];
    O #tIL.Source[8];
    O #tIL.Source[9];
    O #tIL.Source[10];
    O #tIL.Source[11];
    O #tIL.Source[12];
    O #tIL.Source[13];
    O #tIL.Source[14];
    = #tIL.INTERLOCK;

NETWORK
TITLE = Item 40 DV1121 : Update the instance data
    //------------------------------------------------------------------------//
    // Update the instance DB with the calculated interlock flags:            //
    //------------------------------------------------------------------------//
    CALL MOVE
    {value_type := 'Variant'}
    (   IN                   := #tIL ,
        OUT                  := #p[40]
    );

NETWORK
TITLE = Item 41 DV1135 : SMFLx filter outlet drain valve initialise variables
    //------------------------------------------------------------------------//
    // CRITICAL INTERLOCK   CRITICAL INTERLOCK   CRITICAL INTERLOCK   CRITICA //
    // CRITICAL INTERLOCK   CRITICAL INTERLOCK   CRITICAL INTERLOCK   CRITICA //
    //                                                                        //
    // Clear the interlock flag:                                              //
    //------------------------------------------------------------------------//
    A "alwaysLow";
    = #tIL.INTERLOCK;

    //------------------------------------------------------------------------//
    // Clear all interlock values to initialise them to off:                  //
    //------------------------------------------------------------------------//
    CALL FILL_BLK
    {value_type := 'Bool', count_type := 'UInt'}
    (   IN                   := 0 ,
        COUNT                := 15 ,
        OUT                  := #tIL.Source[0]
    );


NETWORK
TITLE = Item 41 DV1135 interlock source : AN ZSC1111 MMFLx Filtration Inlet Flowpath Indicator IN   AN ZSC1109 SMFLx Filtration Line outlet Flowpath Indicator IN
    //------------------------------------------------------------------------//
    // Calculate the interlock condition:                                     //
    //------------------------------------------------------------------------//
    AN(;
    L "idbZSC2".f[4].p.read.mc.STATE;
    L "dbCONST".BLK.ZSC2.STATE.IN;
    ==I;
    );
AN(;
    L "idbZSC2".f[3].p.read.mc.STATE;
    L "dbCONST".BLK.ZSC2.STATE.IN;
    ==I;
    );
    = #tIL.Source[0];

NETWORK
TITLE = Item 41 DV1135 interlock source : A RD1101 Vessel Burst Disc ALARM
    //------------------------------------------------------------------------//
    // Calculate the interlock condition:                                     //
    //------------------------------------------------------------------------//
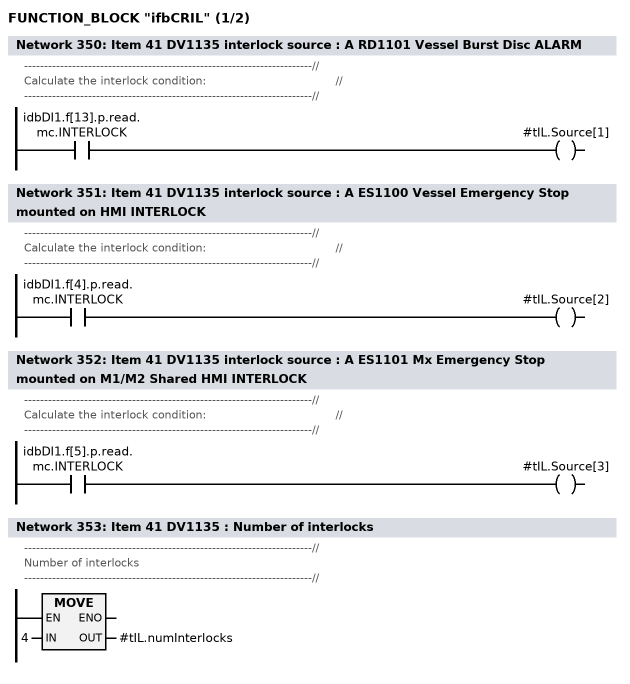
    A idbDI1.f[13].p.read.mc.INTERLOCK;
    = #tIL.Source[1];

NETWORK
TITLE = Item 41 DV1135 interlock source : A ES1100 Vessel Emergency Stop mounted on HMI INTERLOCK
    //------------------------------------------------------------------------//
    // Calculate the interlock condition:                                     //
    //------------------------------------------------------------------------//
    A idbDI1.f[4].p.read.mc.INTERLOCK;
    = #tIL.Source[2];

NETWORK
TITLE = Item 41 DV1135 interlock source : A ES1101 Mx Emergency Stop mounted on M1/M2 Shared HMI INTERLOCK
    //------------------------------------------------------------------------//
    // Calculate the interlock condition:                                     //
    //------------------------------------------------------------------------//
    A idbDI1.f[5].p.read.mc.INTERLOCK;
    = #tIL.Source[3];


NETWORK
TITLE = Item 41 DV1135 : Number of interlocks
    //------------------------------------------------------------------------//
    // Number of interlocks
    //------------------------------------------------------------------------//
    L 4;
    T #tIL.numInterlocks;

NETWORK
TITLE = Item 41 DV1135 : Aggregate individual interlocks into overall INTERLOCK flag
    //------------------------------------------------------------------------//
    // Determine if an interlock is raised:                                   //
    //------------------------------------------------------------------------//
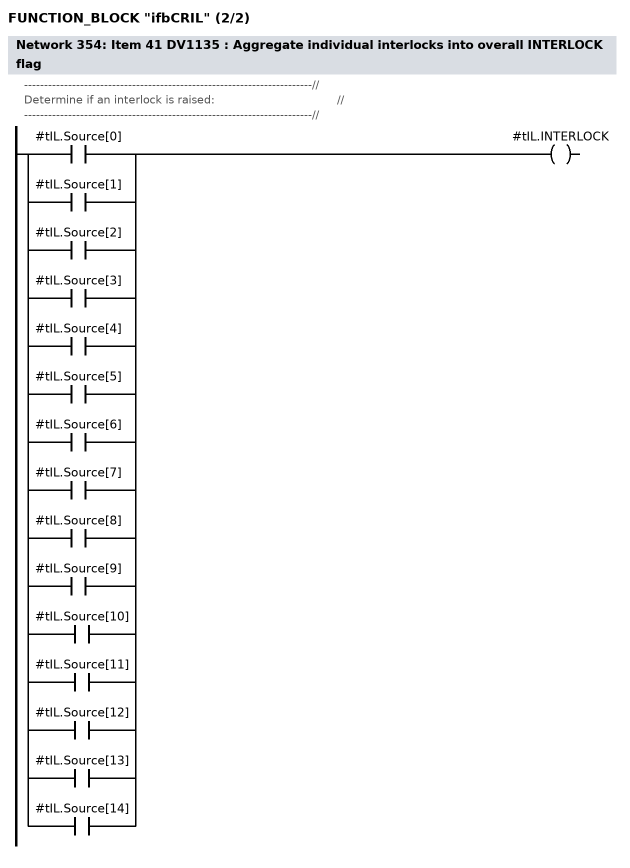
    O #tIL.Source[0];
    O #tIL.Source[1];
    O #tIL.Source[2];
    O #tIL.Source[3];
    O #tIL.Source[4];
    O #tIL.Source[5];
    O #tIL.Source[6];
    O #tIL.Source[7];
    O #tIL.Source[8];
    O #tIL.Source[9];
    O #tIL.Source[10];
    O #tIL.Source[11];
    O #tIL.Source[12];
    O #tIL.Source[13];
    O #tIL.Source[14];
    = #tIL.INTERLOCK;

NETWORK
TITLE = Item 41 DV1135 : Update the instance data
    //------------------------------------------------------------------------//
    // Update the instance DB with the calculated interlock flags:            //
    //------------------------------------------------------------------------//
    CALL MOVE
    {value_type := 'Variant'}
    (   IN                   := #tIL ,
        OUT                  := #p[41]
    );

NETWORK
TITLE = Item 42 DV1137 : SMFLx filter outlet valve initialise variables
    //------------------------------------------------------------------------//
    // CRITICAL INTERLOCK   CRITICAL INTERLOCK   CRITICAL INTERLOCK   CRITICA //
    // CRITICAL INTERLOCK   CRITICAL INTERLOCK   CRITICAL INTERLOCK   CRITICA //
    //                                                                        //
    // Clear the interlock flag:                                              //
    //------------------------------------------------------------------------//
    A "alwaysLow";
    = #tIL.INTERLOCK;

    //------------------------------------------------------------------------//
    // Clear all interlock values to initialise them to off:                  //
    //------------------------------------------------------------------------//
    CALL FILL_BLK
    {value_type := 'Bool', count_type := 'UInt'}
    (   IN                   := 0 ,
        COUNT                := 15 ,
        OUT                  := #tIL.Source[0]
    );


NETWORK
TITLE = Item 42 DV1137 interlock source : AN ZSC1111 MMFLx Filtration Inlet Flowpath Indicator IN   AN ZSC1109 SMFLx Filtration Line outlet Flowpath Indicator IN
    //------------------------------------------------------------------------//
    // Calculate the interlock condition:                                     //
    //------------------------------------------------------------------------//
    AN(;
    L "idbZSC2".f[4].p.read.mc.STATE;
    L "dbCONST".BLK.ZSC2.STATE.IN;
    ==I;
    );
AN(;
    L "idbZSC2".f[3].p.read.mc.STATE;
    L "dbCONST".BLK.ZSC2.STATE.IN;
    ==I;
    );
    = #tIL.Source[0];

NETWORK
TITLE = Item 42 DV1137 interlock source : A RD1101 Vessel Burst Disc ALARM
    //------------------------------------------------------------------------//
    // Calculate the interlock condition:                                     //
    //------------------------------------------------------------------------//
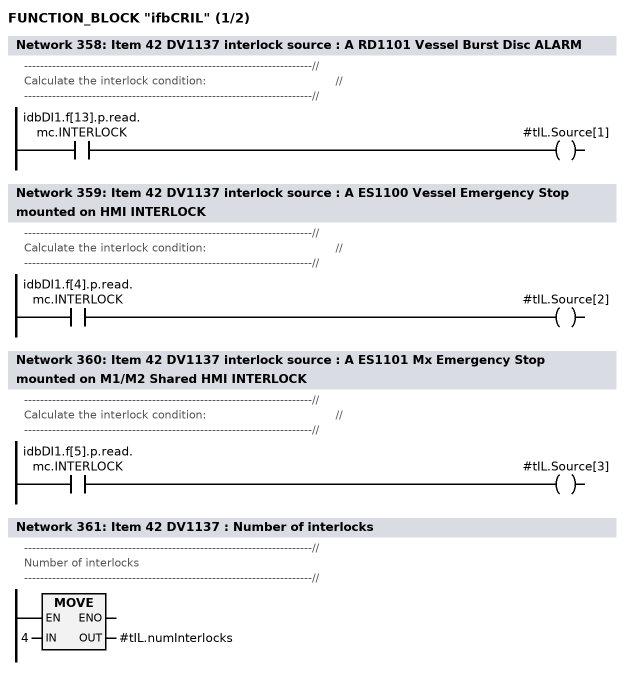
    A idbDI1.f[13].p.read.mc.INTERLOCK;
    = #tIL.Source[1];

NETWORK
TITLE = Item 42 DV1137 interlock source : A ES1100 Vessel Emergency Stop mounted on HMI INTERLOCK
    //------------------------------------------------------------------------//
    // Calculate the interlock condition:                                     //
    //------------------------------------------------------------------------//
    A idbDI1.f[4].p.read.mc.INTERLOCK;
    = #tIL.Source[2];

NETWORK
TITLE = Item 42 DV1137 interlock source : A ES1101 Mx Emergency Stop mounted on M1/M2 Shared HMI INTERLOCK
    //------------------------------------------------------------------------//
    // Calculate the interlock condition:                                     //
    //------------------------------------------------------------------------//
    A idbDI1.f[5].p.read.mc.INTERLOCK;
    = #tIL.Source[3];


NETWORK
TITLE = Item 42 DV1137 : Number of interlocks
    //------------------------------------------------------------------------//
    // Number of interlocks
    //------------------------------------------------------------------------//
    L 4;
    T #tIL.numInterlocks;

NETWORK
TITLE = Item 42 DV1137 : Aggregate individual interlocks into overall INTERLOCK flag
    //------------------------------------------------------------------------//
    // Determine if an interlock is raised:                                   //
    //------------------------------------------------------------------------//
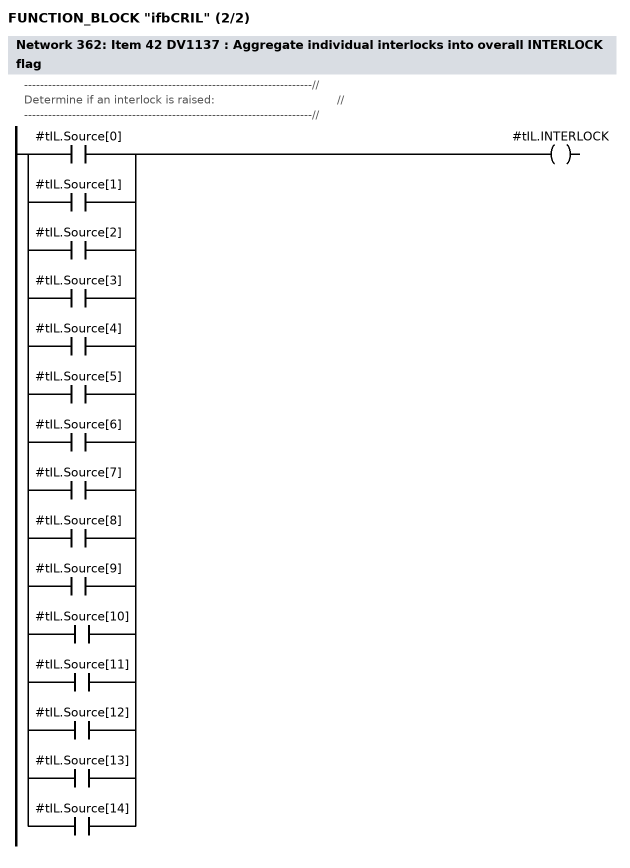
    O #tIL.Source[0];
    O #tIL.Source[1];
    O #tIL.Source[2];
    O #tIL.Source[3];
    O #tIL.Source[4];
    O #tIL.Source[5];
    O #tIL.Source[6];
    O #tIL.Source[7];
    O #tIL.Source[8];
    O #tIL.Source[9];
    O #tIL.Source[10];
    O #tIL.Source[11];
    O #tIL.Source[12];
    O #tIL.Source[13];
    O #tIL.Source[14];
    = #tIL.INTERLOCK;

NETWORK
TITLE = Item 42 DV1137 : Update the instance data
    //------------------------------------------------------------------------//
    // Update the instance DB with the calculated interlock flags:            //
    //------------------------------------------------------------------------//
    CALL MOVE
    {value_type := 'Variant'}
    (   IN                   := #tIL ,
        OUT                  := #p[42]
    );

NETWORK
TITLE = Item 43 DV1171 : MMFLx filter inlet drain valve initialise variables
    //------------------------------------------------------------------------//
    // CRITICAL INTERLOCK   CRITICAL INTERLOCK   CRITICAL INTERLOCK   CRITICA //
    // CRITICAL INTERLOCK   CRITICAL INTERLOCK   CRITICAL INTERLOCK   CRITICA //
    //                                                                        //
    // Clear the interlock flag:                                              //
    //------------------------------------------------------------------------//
    A "alwaysLow";
    = #tIL.INTERLOCK;

    //------------------------------------------------------------------------//
    // Clear all interlock values to initialise them to off:                  //
    //------------------------------------------------------------------------//
    CALL FILL_BLK
    {value_type := 'Bool', count_type := 'UInt'}
    (   IN                   := 0 ,
        COUNT                := 15 ,
        OUT                  := #tIL.Source[0]
    );


NETWORK
TITLE = Item 43 DV1171 interlock source : AN ZSC1113 MMFLx Filtration Inlet Flowpath Indicator IN   AN ZSC1115 MMFLx Filtration Inlet CIP & SIP Flowpath Indicator IN
    //------------------------------------------------------------------------//
    // Calculate the interlock condition:                                     //
    //------------------------------------------------------------------------//
    AN(;
    L "idbZSC2".f[5].p.read.mc.STATE;
    L "dbCONST".BLK.ZSC2.STATE.IN;
    ==I;
    );
AN(;
    L "idbZSC2".f[6].p.read.mc.STATE;
    L "dbCONST".BLK.ZSC2.STATE.IN;
    ==I;
    );
    = #tIL.Source[0];

NETWORK
TITLE = Item 43 DV1171 interlock source : AN ZSC1115 MMFLx Filtration Inlet CIP & SIP Flowpath Indicator IN
    //------------------------------------------------------------------------//
    // Calculate the interlock condition:                                     //
    //------------------------------------------------------------------------//
    AN(;
    L "idbZSC2".f[6].p.read.mc.STATE;
    L "dbCONST".BLK.ZSC2.STATE.IN;
    ==I;
    );
    = #tIL.Source[1];

NETWORK
TITLE = Item 43 DV1171 interlock source : A RD1101 Vessel Burst Disc ALARM
    //------------------------------------------------------------------------//
    // Calculate the interlock condition:                                     //
    //------------------------------------------------------------------------//
